PROGRAM P_RestoreCurrentLanguage
VAR
	waitTon:TON;
	langDone:bool := FALSE;
END_VAR

waitTon(IN:=NOT langDone, PT:=T#8S);

IF waitTon.Q AND NOT langDone THEN
	langDone := TRUE;
	
	//MAIN.M_Log(reqLevel:=CVL.INFO, objectName:= 'P_RestoreCurrentLanguage', sMsg:=RVL.currLanguage, errNo:= 0);
	
	IF RVL.currLanguage <> '' THEN
		VisuElems.CurrentLanguage := RVL.currLanguage;
	ELSE
		VisuElems.CurrentLanguage := 'de';
	END_IF
	
	MAIN.M_Log(reqLevel:=CVL.INFO, objectName:= 'P_RestoreCurrentLanguage', sMsg:= CONCAT('Language = ', RVL.currLanguage), errNo:= 0);
END_IF

END_PROGRAM

(* stored: Version 1.1.0.1, ProductVersion 3.1.4024.3
   POU P_RestoreCurrentLanguage: Id {6123947d-e19f-4e88-b2d7-1ce19cf3fc3d}, SpecialFunc None *)
